//{attribute 'qualified_only'}
VAR_GLOBAL
	robotLeft, robotRight : Robot;
	
	skidLeft, skidRight : MaterialStorage;
	
	stagingTemplateLeft, stagingTemplateRight : WoodBunkTable;
	stagingTableLeft, stagingTableRight : WoodBunkTable;
	magazineLeft, magazineRight : MaterialStorage;
	
	strapper : StrapMachine;
	
	insertionLeft, insertionRight : PneumaticInsertionEIP;	
	insertionBottom : AirPiston;
	
	topSuction : ARRAY[1..3] OF SuctionPad;
	leftSuction : ARRAY[1..4] OF SuctionPad;
	rightSuction : ARRAY[1..4] OF SuctionPad; 
	bottomSuction : ARRAY[1..2] OF SuctionPad;
	
	toolStorageLeft, toolStorageRight : A21ToolStorage;
END_VAR

(* stored: Version 1.1.0.1, ProductVersion 3.1.4024.11
   GVL Hardware: Id {72ad6a3a-e035-4ae1-b9b7-c68bdd948b2f} *)
